FUNCTION_BLOCK AX_OR_4 (* FB to calculate boolean OR *)
  (* Standard: 61499-2; Description: Copyright (c) 2024 HR Agrartechnik GmbH This program and the accompanying materials are made available under the terms of the Eclipse Public License 2.0 which is available at https://www.eclipse.org/legal/epl-2.0/ SPDX-License-Identifier: EPL-2.0 *)
  (* Version 1.0, 2024-10-23, franz *)
  PACKAGE io::adp::boolean;
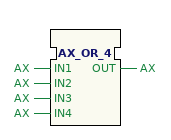
  SOCKETS
    IN1 : AX; (* OR input 1 *)
    IN2 : AX; (* OR input 2 *)
    IN3 : AX; (* OR input 3 *)
    IN4 : AX; (* OR input 4 *)
  END_SOCKETS
  PLUGS
    OUT : AX; (* OR result *)
  END_PLUGS
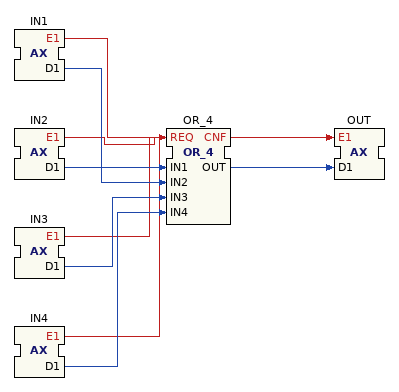
  FBS
    OR_4 : OR_4;
  END_FBS
  EVENT_CONNECTIONS
    IN1.E1 TO OR_4.REQ;
    IN2.E1 TO OR_4.REQ;
    OR_4.CNF TO OUT.E1;
    IN3.E1 TO OR_4.REQ;
    IN4.E1 TO OR_4.REQ;
  END_CONNECTIONS
  DATA_CONNECTIONS
    IN1.D1 TO OR_4.IN1;
    IN2.D1 TO OR_4.IN2;
    OR_4.OUT TO OUT.D1;
    IN3.D1 TO OR_4.IN3;
    IN4.D1 TO OR_4.IN4;
  END_CONNECTIONS
END_FUNCTION_BLOCK
